FUNCTION_BLOCK ABSTRACT Body_Task_Base
VAR
	_busy : BOOL;
	_error : BOOL;
	_done : BOOL;
END_VAR

METHOD Abort : BOOL
VAR_INPUT
END_VAR
END_METHOD

PROPERTY Busy : bool
GET
Busy := _busy;
END_GET
END_PROPERTY

PROPERTY Done : bool
GET
Done := _done;
END_GET
END_PROPERTY

PROPERTY Error : bool
GET
Error := _error;
END_GET
END_PROPERTY

END_FUNCTION_BLOCK

(* stored: Version 1.1.0.1, ProductVersion 3.1.4024.11
   POU Body_Task_Base: Id {5206f1e1-b365-4cd6-8c6b-727542dc36a0}, SpecialFunc None
   Method Abort: Id {7682a0d7-7f5f-4e3b-b408-a481c1361e56}
   Property Busy: Id {c817590d-4e06-4806-9fe4-aec253cd45ec}
   Get Get: Id {cd5751fb-3e1c-4787-b81c-e4b5122e22eb}
   Property Done: Id {3902f8bd-04d2-475a-b6f5-7ad516e9e0b0}
   Get Get: Id {6135de80-e2c8-4195-821d-76f1832038cf}
   Property Error: Id {379fa651-c821-4d8c-a2b7-dafbbf5ffda5}
   Get Get: Id {a47ead4a-09de-41a4-8d64-457e75596e0c} *)
